INTERFACE ICUTask

PROPERTY Task : REFERENCE TO TcoCore.TcoTask
GET
END_GET
END_PROPERTY

END_INTERFACE

(* stored: Version 1.1.0.1, ProductVersion 3.1.4024.9
   Itf ICUTask: Id {343605ca-9899-4f92-af75-d6c9f6962b10}
   Property Task: Id {79c92659-cce6-4fd1-8646-993eb5b2eb99}
   Get Get: Id {4770c50c-d51e-4d68-855b-885130702611} *)
